PROGRAM Examples

//PointerExample();
//ReferenceExample();
InterfaceExample();

END_PROGRAM

(* stored: Version 1.1.0.1, ProductVersion 3.1.4024.10
   POU Examples: Id {87525701-b5c6-4916-893e-373055ab34e3}, SpecialFunc None *)
